TEXTLIST FadeTime
  0 = 'Extended Fade Time'
  1 = '0,7 s'
  2 = '1,0 s'
  3 = '1,4 s'
  4 = '2,0 s'
  5 = '2,8 s'
  6 = '4,0 s'
  7 = '5,7 s'
  8 = '8,0 s'
  9 = '11,3 s'
  10 = '16,0 s'
  11 = '22,6 s'
  12 = '32,0 s'
  13 = '45,3 s'
  14 = '64,0 s'
  15 = '90,5 s'
   = ''
END_TEXTLIST

(* stored: Version 1.1.0.1, ProductVersion 3.1.4024.4
   TextList FadeTime: Id {22c4f2cc-31c3-4afc-8c1f-b4dd2efe8f10} *)
